(* CODESYS project Uppgift-15.project

Project tree, tasks and I/O mapping:
  Device : CODESYS Control Win V3, 3S - Smart Software Solutions GmbH, order no. 305021, version 3.5.10.40
    application Application
      libraries: Standard, * (System)
      task MainTask (cyclic, interval t#20ms, priority 1) calls PLC_PRG
      program PLC_PRG [ST]
      global variables GVL
      Symbols
*)

// Device/Application/GVL
{attribute 'qualified_only'}
VAR_GLOBAL
	// Sensors.
	// Input Conveyor
	SensorDrop: BOOL; // Systeminput sensor
	Sensor1: BOOL; // Conveor 1. wait for rotationtable conveyor
	
	
	//Rotatinal  Conveoyr. boc ontop
	Sensor2: BOOL; // Rotation signal. Conecteed to conveor 2 input/droopin conveor.
	Sensor3: BOOL; // Rotation conveor. insignal 
	
	//Rotation sensor. convey direction
	Sensor4: BOOL; // Rotation signal. Conecteed to conveor 3 Output conveor.
	Sensor5: BOOL; // Rotation conveor. box on conveor
	
	// conveyor 3 output
	Sensor6: BOOL; // Conveor 3. Output conveour. box ontop.
	
	
	// Conveyor movment.
	Motor1Fwd: BOOL; // Conveor 1 motor.
	Motor2Fwd: BOOL; // Conveor 2 motor. Rotational Conveor table
	Motor3Fwd: BOOL; // Conveor 3 motor. Output conveour.
	
	// Conveyor movment
	TurnFwd: BOOL; // Turn conveor 2 to conveor 3 Output conveor.
	TurnRev: BOOL; // Turn conveor 2 to conveor 1 input/droopin conveor.
END_VAR

// Device/Application/PLC_PRG
PROGRAM PLC_PRG
VAR
	stateCase: int;
END_VAR



CASE stateCase OF
	0: // Listening
	IF(gvl.SensorDrop) THEN
		stateCase := 1;
	END_IF
	1: // Move to rotational movement
	gvl.Motor1Fwd := TRUE;
	
	IF gvl.Sensor1 THEN
		gvl.Motor1Fwd := FALSE;
		stateCase := 2;
	END_IF
	
	2: // Rotationcheck
	IF gvl.Sensor4 THEN
		gvl.TurnRev := FALSE;
		
		IF gvl.Sensor3 THEN
			gvl.Motor2Fwd 	:= FALSE;
			gvl.Motor1Fwd 	:= FALSE;
			stateCase 		:= 3;
		ELSE
			gvl.Motor2Fwd 	:= TRUE;
			gvl.Motor1Fwd 	:= TRUE;
		END_IF
	ELSE
		gvl.TurnRev := TRUE;
	END_IF
	
	3: // Turn Converour check
	IF gvl.Sensor3 THEN
		IF gvl.Sensor5 = FALSE THEN
			gvl.TurnFwd := TRUE;
		ELSE
			gvl.TurnFwd := FALSE;
			stateCase := 4;
		END_IF
	ELSE
		stateCase := 0;
	END_IF
	
	4: // Movebox to conveor 3.
	IF gvl.Sensor6 = FALSE THEN
		gvl.Motor3Fwd := TRUE;
		gvl.Motor2Fwd := TRUE;
		ELSE
			gvl.Motor3Fwd := FALSE;
			gvl.Motor2Fwd := FALSE;
			stateCase := 5;
	END_IF
	
	5: // Reset conveyor 2 rotational
	
	IF gvl.Sensor4 = FALSE THEN
		gvl.TurnRev := TRUE;
	ELSE
		gvl.TurnRev := FALSE;
		stateCase := 0;
	END_IF
END_CASE

END_PROGRAM
